Yaskawa INFORM job: R2_O5(90,-90).JBI

/JOB
//NAME R2_O5(90,-90)
///FOLDERNAME PROGRAMY_TESTOWE_ODWLOK
//POS
///NPOS 26,26,26,2,0,0
///TOOL 0
///POSTYPE PULSE
///PULSE
C00000=-120667,124465,54470,-40687,78894,74346
C00001=-120667,122061,54158,-40809,78093,74661
C00002=-120667,121136,54084,-40862,77763,74791
C00003=-120667,121750,53626,-40789,78221,74611
C00004=-120051,121151,54106,-41153,78011,74935
C00005=-120667,121771,54124,-40643,79250,74206
C00006=-120667,123465,54293,-40248,82775,72848
C00007=-120667,124707,54470,-40065,85755,71718
C00008=-120667,125542,54613,-40015,88183,70803
C00009=-120667,126507,54799,-40125,92344,69239
C00010=-120667,126430,54783,-40163,92737,69084
C00011=-120667,126842,54869,-40358,94967,68230
C00012=-120668,127920,55123,-40391,95274,68112
C00013=-120668,130710,55896,-40475,96012,67826
C00014=-132474,154538,69486,-38780,96231,64957
C00015=-132464,135192,59707,-38494,93134,66082
C00016=-133927,132367,58821,-37901,91869,66005
C00017=-134512,131314,58578,-37666,91339,65980
C00018=-135314,132040,59603,-37355,90835,65866
C00019=-134512,131314,58578,-37666,91339,65980
C00020=-133380,129585,56818,-38097,91916,66186
C00021=-133402,127481,55619,-38076,91635,66277
C00022=-133380,129585,56818,-38097,91916,66186
C00023=-132793,130667,57098,-38334,92440,66211
C00024=-131326,133560,58070,-38930,93693,66288
C00025=-131336,152603,67346,-39259,96892,65107
BC00000=138013,629359,1075175
BC00001=132399,630740,1075175
BC00002=130154,631293,1075175
BC00003=130154,631293,1075175
BC00004=130154,631293,1075175
BC00005=130165,633198,1075175
BC00006=130154,643507,1075175
BC00007=130145,651198,1075175
BC00008=130132,662347,1075175
BC00009=130094,677048,1075175
BC00010=130110,680055,1075175
BC00011=130112,686079,1075175
BC00012=132357,686288,1075175
BC00013=137971,686811,1075175
BC00014=189432,689442,1075175
BC00015=189432,689442,1075175
BC00016=189432,689442,1075175
BC00017=189432,689442,1075175
BC00018=189432,689442,1075175
BC00019=189432,689442,1075175
BC00020=189432,689442,1075175
BC00021=189432,689442,1075175
BC00022=189432,689442,1075175
BC00023=189432,689442,1075175
BC00024=189432,689442,1075175
BC00025=189432,689442,1075175
EC00000=798156,-556475
EC00001=798156,-556475
EC00002=798156,-556475
EC00003=798156,-556475
EC00004=798156,-556475
EC00005=798156,-556475
EC00006=798156,-556475
EC00007=798156,-556475
EC00008=798156,-556475
EC00009=798156,-556475
EC00010=798156,-556475
EC00011=798156,-556475
EC00012=798156,-556475
EC00013=798156,-556475
EC00014=798156,-556475
EC00015=798156,-556475
EC00016=798156,-556475
EC00017=798156,-556475
EC00018=798156,-556475
EC00019=798156,-556475
EC00020=798156,-556475
EC00021=798156,-556475
EC00022=798156,-556475
EC00023=798156,-556475
EC00024=798156,-556475
EC00025=798156,-556475
///POSTYPE BASE
///RECTAN
///RCONF 0,0,0,0,0,0,0,0,0,0,0,0,0,0,0,0,0,0,0,0,0,0,0,0
P00006=0.222,-3.123,-1.508,0.0000,0.0000,0.0000
P00021=-0.225,-6.128,-0.405,0.0000,0.0000,0.0000
//INST
///DATE 2023/11/22 16:04
///ATTR SC,RW
///GROUP1 RB1,BS1
///GROUP2 ST1
NOP
'r2_O5(90,-90)
'Path W1199
SSFTOF
SSFTON P021
MOVJ C00000 BC00000 VJ=100.00  +MOVJ EC00000 VJ=100.00
SMOVL C00001 BC00001 V=400.0  +MOVJ EC00001
SMOVL C00002 BC00002 V=100.0 PL=0  +MOVJ EC00002
SREFP 1 C00003 BC00003  +REFP EC00003
SREFP 2 C00004 BC00004  +REFP EC00004
MACRO1 MJ#(0) ARGF0
ARCON
SMOVL C00005 BC00005 V=10.0  +MOVJ EC00005
SMOVL C00006 BC00006 V=10.0  +MOVJ EC00006
SMOVC C00007 BC00007 V=10.0  +MOVJ EC00007
SMOVC C00008 BC00008 V=10.0  +MOVJ EC00008
SMOVC C00009 BC00009 V=10.0 FPT  +MOVJ EC00009
SMOVC C00010 BC00010 V=10.0  +MOVJ EC00010
SMOVC C00011 BC00011 V=10.0 FPT  +MOVJ EC00011
ARCOF
SMOVL C00012 BC00012 V=400.0  +MOVJ EC00012
SMOVL C00013 BC00013 V=1000.0  +MOVJ EC00013
SSFTOF
'Path S1205
SSFTOF
MOVJ C00014 BC00014 VJ=100.00  +MOVJ EC00014 VJ=100.00
MOVJ C00015 BC00015 VJ=100.00  +MOVJ EC00015 VJ=100.00
MOVL C00016 BC00016 V=400.0  +MOVJ EC00016 VJ=100.00
SMOVL C00017 BC00017 V=60.0  +MOVJ EC00017
SREFP 3 C00018 BC00018  +REFP EC00018
CALL JOB:SEARCH-R1-S1
SET P021 P006
SSFTON P021
SMOVL C00019 BC00019 V=60.0  +MOVJ EC00019
SMOVL C00020 BC00020 V=60.0  +MOVJ EC00020
SREFP 3 C00021 BC00021  +REFP EC00021
CALL JOB:SEARCH-R1-S1
SET P021 P006
SSFTON P021
SMOVL C00022 BC00022 V=60.0  +MOVJ EC00022
MOVL C00023 BC00023 V=400.0  +MOVJ EC00023 VJ=100.00
MOVL C00024 BC00024 V=1000.0  +MOVJ EC00024 VJ=100.00
MOVL C00025 BC00025 V=1000.0  +MOVJ EC00025 VJ=100.00
END
